Fanuc TP program (LS listing): at_pick.ls

/PROG  AT_PICK
/ATTR
COMMENT		= "";
DEFAULT_GROUP	= 1,*,*,*,*;
/MN
 : UFRAME_NUM=1 ;
 : UTOOL_NUM=1 ;
 : PR[2:LPOS]=LPOS ;
 : IF (PR[2,1]<(-100)),JMP LBL[500] ;
 : IF (PR[2,1]<100),JMP LBL[500] ;
 : IF (PR[2,2]<(-100)),JMP LBL[500] ;
 : IF (PR[2,2]<100),JMP LBL[500] ;
 : IF (PR[2,3]<(-100)),JMP LBL[500] ;
 : IF (PR[2,3]<300),JMP LBL[500] ;
 : R[2:zoneID]=1 ;
 : END ;
 :  ;
 : LBL[500] ;
 :   R[2:zoneID]=0 ;
 :   END ;
/POS
/END
